FUNCTION F_GetFunctionDataEmulation : ST_FunctionDataEmulation;
(**************************************************************************************
 * 	Application		:	BoxControl Framework
 *	Revision		:	$Revision: 404529 $
 *	Revision date	:	$Date: 2018-04-23 08:21:38 +0200 (Mo., 23 Apr 2018) $
 *	Last changed by	:	$Author: b7bolm $
 *	URL				:	$URL: http://almscdc.swisslog.com/repo/SWPD/Development/BoxControlFramework/20_Release/trunk/01_Software/BCF/BCF/JumpStart/20_Product/11_Emu/12_E_Functions/10_Lib/10_Conv/10_Functions/F_GetFunctionDataEmulation.TcPOU $
 *
 *	Purpose			:	Returns function data
 *
 * ------------------------------------------------------------------------------------
 *	Copyright Swisslog [IP AG], Switzerland. All rights reserved.
 * 
 * ------------------------------------------------------------------------------------
 *	
 * 	Revision History: 
 *
 * 	VERSION			DATE			INITIALS			DESCRIPTION
 *	0.1				01.01.2001		swl					Example
 *
 **************************************************************************************)
VAR_INPUT
	eFunctionNumber		: E_FunctionNumber; // Element function Number
END_VAR


// Check if function number is valid
IF eFunctionNumber > E_FunctionNumber.F_BEGIN_FUNCTION AND
   eFunctionNumber < E_FunctionNumber.F_END_FUNCTION THEN

   // Check reference is valid
   IF __ISVALIDREF(FunctionRegistryEmulation[eFunctionNumber].rFunction) THEN
	   
   		// Return function data emulation
   		F_GetFunctionDataEmulation := FunctionRegistryEmulation[eFunctionNumber].rFunction.FunctionData;
   END_IF
END_IF

END_FUNCTION

(* stored: Version 1.1.0.1, ProductVersion 3.1.4022.12
   POU F_GetFunctionDataEmulation: Id {e188cb39-a85f-4407-b8c0-de272dc46b69}, SpecialFunc None *)
